// TIA Portal project "LiveTwin_Pump" (V17)

(* hardware
DEVICE "S7-1200 station_1"  S7-1200 Station
   slot 0: "Rack_0"  S7-1200 Rack  Rack  V1.0
   slot 1: "PLC_1"  CPU 1212C DC/DC/DC  6ES7 212-1AE40-0XB0  V4.4
*)

// ===== PLC "PLC_1"  CPU 1212C DC/DC/DC =====

VAR_GLOBAL   // PLC tag table "Default tag table"
   "Manipulator" AT %MW0 : Int;
END_VAR

VAR_GLOBAL CONSTANT   // PLC tag table "Default tag table"
   "STATE_FILL_TANK" : Int := 1;
   "STATE_HEAT_TANK" : Int := 2;
   "STATE_FILL_BOTTLE" : Int := 3;
   "STATE_SHIFT_BOTTLE" : Int := 4;
   "STATE_STOP" : Int := 5;
   "STATE_RESET" : Int := 6;
   "STATE_ERROR" : Int := 7;
END_VAR

DATA_BLOCK "LiveTwin_Pump_DB"   // DB61
{ S7_Optimized_Access := 'TRUE' }
VERSION : 0.1
// stored: InstanceOfName LiveTwin_Pump
"LiveTwin_Pump"
BEGIN
END_DATA_BLOCK

DATA_BLOCK "GlobalDB_LiveTwin"   // DB62
{ S7_Optimized_Access := 'TRUE' }
VERSION : 0.1
   VAR
      pump_speed : Real;
      flow_rate_l_min : Real;
   END_VAR
BEGIN
END_DATA_BLOCK

FUNCTION_BLOCK "LiveTwin_Pump"   // FB60, SCL
{ S7_Optimized_Access := 'TRUE' }
VERSION : 0.1
   VAR
      IEC_Timer_0_Instance : TON_TIME;
      "counter" : DInt;
      pump_speed : Real := 2500.0;
      state : USInt;
   END_VAR
   VAR_TEMP
      timer_out : Bool;
      timer_val : Time;
      timer_preset : Time;
      temp_random : Real;
   END_VAR
   VAR CONSTANT
      timer_in : Bool := true;
   END_VAR
BEGIN
   #IEC_Timer_0_Instance(IN := #timer_in,
                         PT := T#10ms,
                         Q => #timer_out,
                         ET => #timer_val);

   IF #timer_out THEN
       #counter := #counter + 1;
       RESET_TIMER(#IEC_Timer_0_Instance);
   END_IF;

   IF #counter >= 500 THEN
       #counter := 0;
       IF #state <= 2 THEN
           #state := #state + 1;
       ELSE
           #state := 0;
       END_IF;
   END_IF;

   "Random_Number"(Min := -1,
                   Max := 1,
                   RandomNumber => #temp_random);

   CASE #state OF
       0:
           #pump_speed := #pump_speed + 0.2;
       1:
           #pump_speed := #pump_speed + #temp_random * 0.2;
       2:
           IF #pump_speed >= 2510 THEN
               #pump_speed := #pump_speed - 0.21;
           END_IF;
       3:
           #pump_speed := #pump_speed + #temp_random * 0.2;
           IF #pump_speed < 2500 THEN
               #pump_speed := 2500;
           END_IF;
   END_CASE;

   "GlobalDB_LiveTwin".pump_speed := #pump_speed;
END_FUNCTION_BLOCK

FUNCTION "Random_Number" : Void   // FC3, SCL
{ S7_Optimized_Access := 'TRUE' }
VERSION : 0.1
   VAR_INPUT
      Min : Int;
      Max : Int;
   END_VAR
   VAR_OUTPUT
      RandomNumber : Int;
   END_VAR
   VAR_TEMP
      range : Int;
      tmp : Int;
      rdsys : DTL;
      ret : Int;
   END_VAR
BEGIN
   // generate random number
   #ret := RD_SYS_T(#rdsys);
   #tmp := UDINT_TO_INT(#rdsys.NANOSECOND);
   IF #tmp < 0 THEN
       #tmp := #tmp * - 1;
   END_IF;

   "Manipulator" := "Manipulator" + 1;

   IF "Manipulator" = 10 THEN
       "Manipulator" := 1;
   END_IF;

   #tmp := #tmp / "Manipulator";

   #range := #Max - #Min;

   #tmp := #tmp MOD (#range + 1);
   #RandomNumber := #tmp + #Min;
END_FUNCTION

ORGANIZATION_BLOCK "Main"   // OB1, LAD, ProgramCycle
TITLE = "Main Program Sweep (Cycle)"
{ S7_Optimized_Access := 'TRUE' }
VERSION : 0.1
   VAR_INPUT
      Initial_Call : Bool;   // Initial call of this OB
      Remanence : Bool;   // =True, if remanent data are available
   END_VAR
BEGIN

REGION Network 1
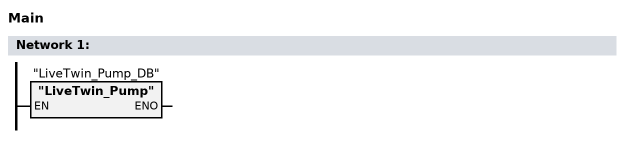
   RUNG wire#powerrail
      "LiveTwin_Pump_DB"()
   END_RUNG
   // the same network as SCL:
   "LiveTwin_Pump_DB"();   // "LiveTwin_Pump"
END_REGION
END_ORGANIZATION_BLOCK